FUNCTION_BLOCK SS4_v_ps02Pub_Sub (* Composite FB wrapping other FBs *)
  (* Standard: 61499-2 *)
  (* Version 1.0, 2024-10-03, DEVIASH *)
  PACKAGE UserLibs::SubStations::SS4;
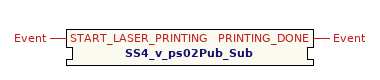
  EVENT_INPUT
    START_LASER_PRINTING; (* Initialization Request *)
  END_EVENT
  EVENT_OUTPUT
    PRINTING_DONE; (* Initialization Confirm *)
  END_EVENT
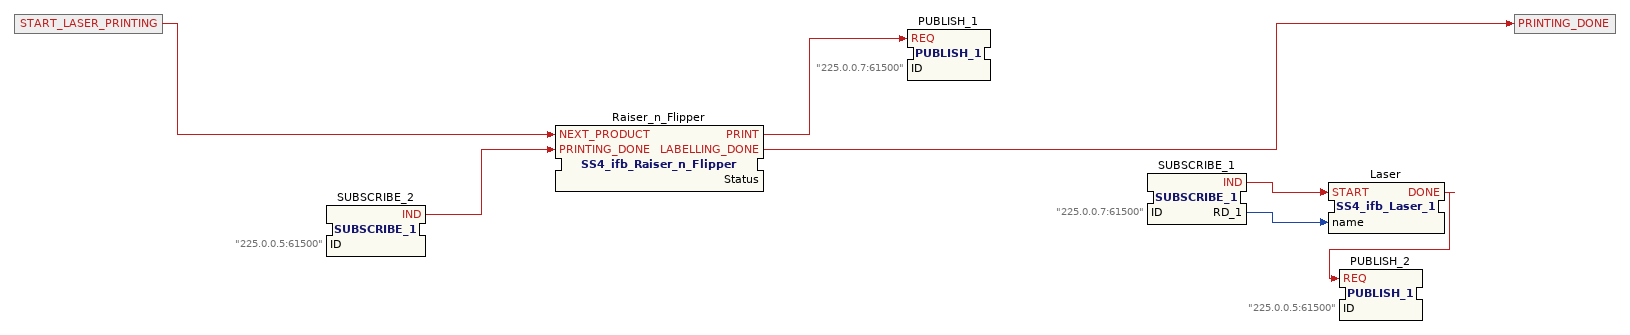
  FBS
    Raiser_n_Flipper : SS4_ifb_Raiser_n_Flipper;
    Laser : SS4_ifb_Laser_1;
    PUBLISH_1 : PUBLISH_1(ID := "225.0.0.7:61500");
    SUBSCRIBE_1 : SUBSCRIBE_1(ID := "225.0.0.7:61500");
    PUBLISH_2 : PUBLISH_1(ID := "225.0.0.5:61500");
    SUBSCRIBE_2 : SUBSCRIBE_1(ID := "225.0.0.5:61500");
  END_FBS
  EVENT_CONNECTIONS
    START_LASER_PRINTING TO Raiser_n_Flipper.NEXT_PRODUCT;
    Laser.DONE TO PUBLISH_2.REQ;
    Raiser_n_Flipper.LABELLING_DONE TO PRINTING_DONE;
    Raiser_n_Flipper.PRINT TO PUBLISH_1.REQ;
    SUBSCRIBE_1.IND TO Laser.START;
    SUBSCRIBE_2.IND TO Raiser_n_Flipper.PRINTING_DONE;
  END_CONNECTIONS
  DATA_CONNECTIONS
    SUBSCRIBE_1.RD_1 TO Laser.name;
  END_CONNECTIONS
END_FUNCTION_BLOCK
